DATA_BLOCK "DB_FB_EFF_TestHarness"
{ S7_Optimized_Access := 'TRUE' }
VERSION : 0.1
   "FB_EFF_TestHarness"
BEGIN
END_DATA_BLOCK
